TYPE ST_GripperManagerState :
STRUCT
    bCommunicationReady : BOOL;
    bHealthy            : BOOL;
    bManualReady        : BOOL;
    bAutoReady          : BOOL;
    bBusy               : BOOL;
    bSimulationActive   : BOOL;
    bStopAcknowledged   : BOOL;
    bStopError          : BOOL;
    udStopErrorCode     : UDINT;
    eOwner              : E_GripperControlOwner;
    eActiveCommand      : E_GripperCommand;
END_STRUCT
END_TYPE

(* stored: Version 1.1.0.1, ProductVersion 3.1.4026.20
   DUT ST_GripperManagerState: Id {8eb730e1-5855-4b68-8fb1-c22975db65c2} *)
